(* PLC project Sin nombre, Desconocido Sin nombre 1 *)
(* stored: creationDateTime 2024-06-17T10:23:13, modificationDateTime 2024-06-20T13:18:59 *)

PROGRAM Paletizador
  VAR
    Inicio AT %IX100.0 : BOOL;
    Paro AT %IX100.1 : BOOL;
    Motor_cinta_Horizontal AT %QX100.0 : BOOL;
    Motor_cinta_Inclinado AT %QX100.1 : BOOL;
    Motor_cinta_Paletizador AT %QX100.2 : BOOL;
    Contador_Cajas AT %IX100.2 : BOOL;
    Piston_1 AT %QX100.3 : BOOL;
    Sensor_Piston_1 AT %IX100.3 : BOOL;
  END_VAR
  VAR
    CTU0 : CTU;
  END_VAR
  VAR
    Piston_Compuerta AT %QX100.4 : BOOL;
    Sensor_Piston_Compuerta AT %IX100.4 : BOOL;
    Compuerta AT %QX100.5 : BOOL;
    Sensor_Compuerta AT %IX100.5 : BOOL;
  END_VAR
  VAR
    CTU1 : CTU;
  END_VAR
  VAR
    Generador_Cajas AT %QX100.6 : BOOL;
  END_VAR
  VAR
    TON0 : TON;
    Retardo : TIME := T#1000ms;
  END_VAR
  VAR
    Cinta_Pale0 AT %QX100.7 : BOOL;
    Cinta_Pale1 AT %QX100.8 : BOOL;
    Generador_pales AT %QX100.9 : BOOL;
    Cinta_Paletizador AT %QX100.10 : BOOL;
    Sensor_Pale_0 AT %IX100.6 : BOOL;
    Sensor_Pale_1 AT %IX100.7 : BOOL;
    limite_altura AT %QX100.12 : BOOL;
    subir_pale AT %QX100.11 : BOOL;
    bajar_pale AT %QX100.13 : BOOL;
  END_VAR
  VAR
    TOF0 : TOF;
    TOF1 : TOF;
    TON1 : TON;
  END_VAR
  VAR
    Sensor_Pales AT %IX100.8 : BOOL;
    sensor_ascensor AT %IX100.9 : BOOL;
  END_VAR
  VAR
    CTU2 : CTU;
    TON2 : TON;
  END_VAR
  VAR
    sensor_bajada AT %IX100.10 : BOOL;
  END_VAR
  VAR
    TON3 : TON;
    TOF2 : TOF;
    TON4 : TON;
  END_VAR
  VAR  (* added by the conversion: wires and edge detectors of the diagram *)
    R_TRIG1 : R_TRIG;
    R_TRIG2 : R_TRIG;
    R_TRIG3 : R_TRIG;
    R_TRIG4 : R_TRIG;
    R_TRIG5 : R_TRIG;
  END_VAR

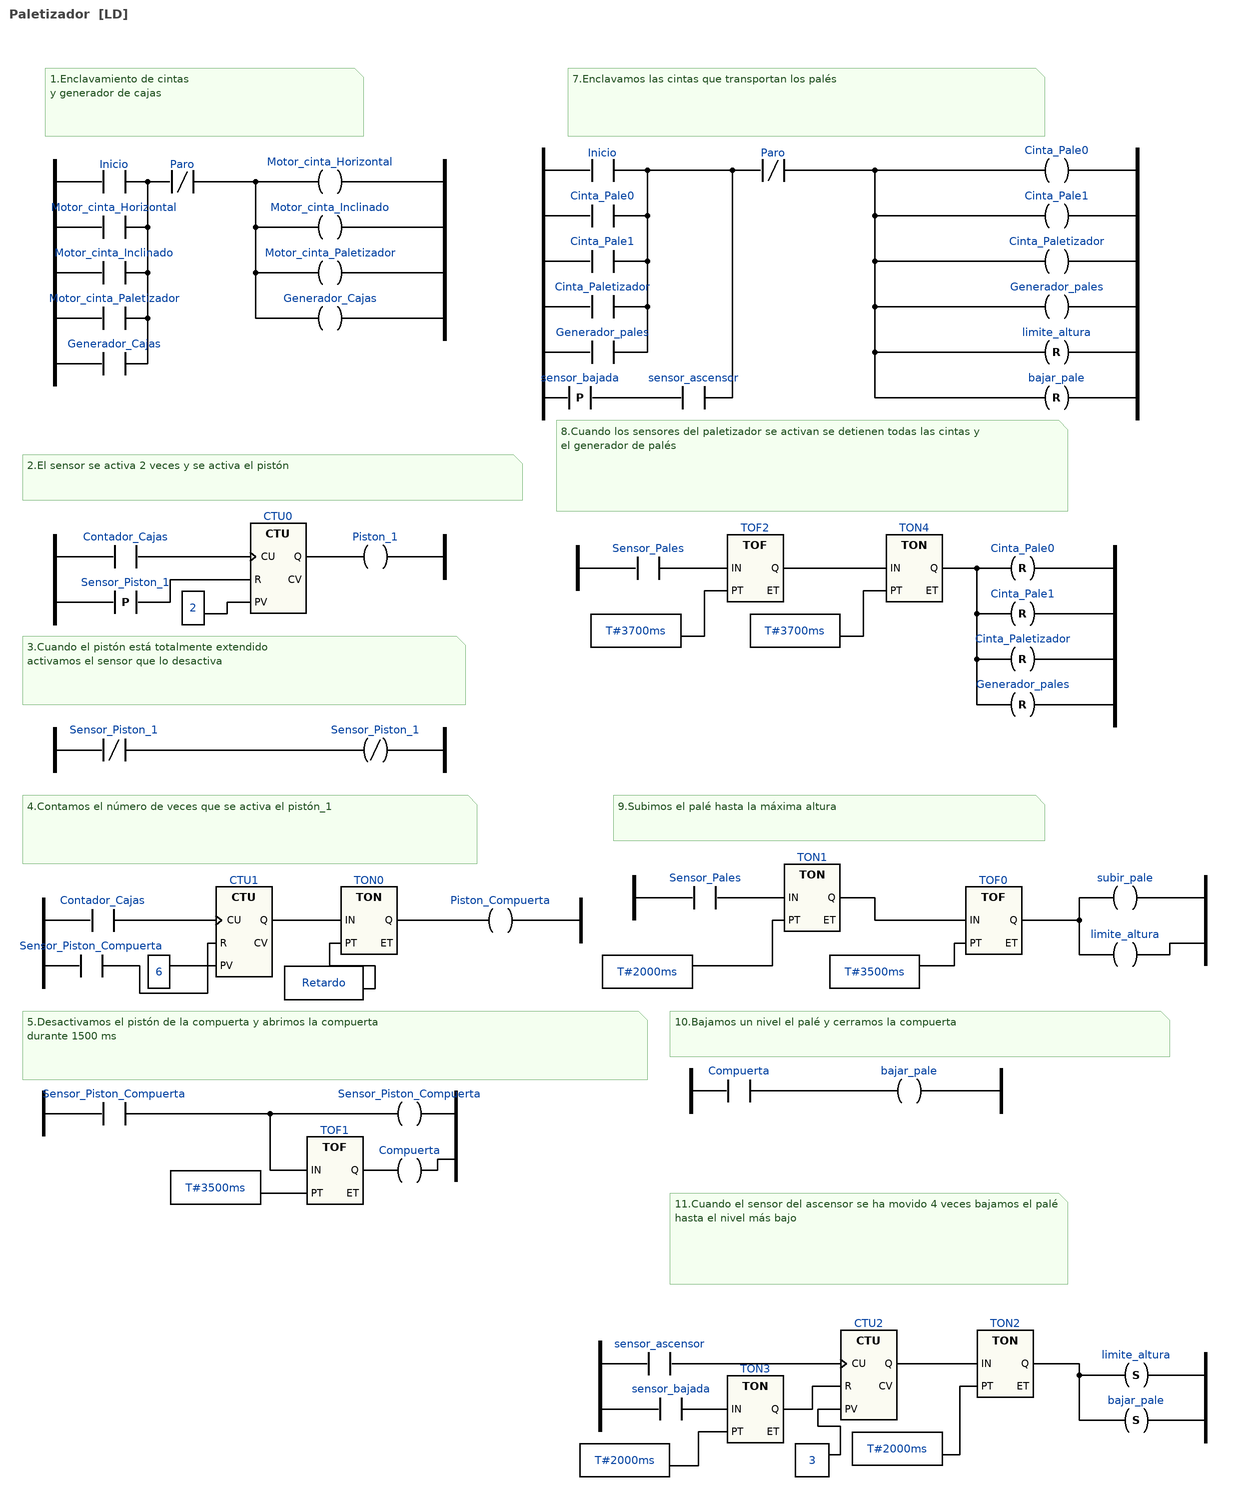
(* LD diagram, written out as Structured Text *)
(* 1.Enclavamiento de cintas
y generador de cajas *)
(* 7.Enclavamos las cintas que transportan los palés *)
Motor_cinta_Horizontal := (Inicio OR Motor_cinta_Horizontal OR Motor_cinta_Inclinado OR Motor_cinta_Paletizador OR Generador_Cajas) AND NOT Paro;
Motor_cinta_Inclinado := (Inicio OR Motor_cinta_Horizontal OR Motor_cinta_Inclinado OR Motor_cinta_Paletizador OR Generador_Cajas) AND NOT Paro;
Motor_cinta_Paletizador := (Inicio OR Motor_cinta_Horizontal OR Motor_cinta_Inclinado OR Motor_cinta_Paletizador OR Generador_Cajas) AND NOT Paro;
(* 8.Cuando los sensores del paletizador se activan se detienen todas las cintas y 
el generador de palés *)
(* 2.El sensor se activa 2 veces y se activa el pistón *)
R_TRIG1(CLK := Contador_Cajas);
R_TRIG2(CLK := Sensor_Piston_1);
CTU0(CU := R_TRIG1.Q, R := R_TRIG2.Q, PV := 2);
Piston_1 := CTU0.Q;
(* 3.Cuando el pistón está totalmente extendido
activamos el sensor que lo desactiva *)
(* 4.Contamos el número de veces que se activa el pistón_1 *)
(* 9.Subimos el palé hasta la máxima altura *)
R_TRIG3(CLK := Contador_Cajas);
CTU1(CU := R_TRIG3.Q, R := Sensor_Piston_Compuerta, PV := 6);
TON0(IN := CTU1.Q, PT := Retardo);
Piston_Compuerta := TON0.Q;
(* 5.Desactivamos el pistón de la compuerta y abrimos la compuerta
durante 1500 ms *)
(* 10.Bajamos un nivel el palé y cerramos la compuerta *)
Sensor_Piston_Compuerta := Sensor_Piston_Compuerta;
Generador_Cajas := (Inicio OR Motor_cinta_Horizontal OR Motor_cinta_Inclinado OR Motor_cinta_Paletizador OR Generador_Cajas) AND NOT Paro;
Sensor_Piston_1 := NOT (NOT Sensor_Piston_1);
TOF1(IN := Sensor_Piston_Compuerta, PT := T#3500ms);
Compuerta := TOF1.Q;
TON1(IN := Sensor_Pales, PT := T#2000ms);
TOF0(IN := TON1.Q, PT := T#3500ms);
subir_pale := TOF0.Q;
limite_altura := TOF0.Q;
bajar_pale := Compuerta;
(* 11.Cuando el sensor del ascensor se ha movido 4 veces bajamos el palé hasta el nivel más bajo *)
R_TRIG4(CLK := sensor_ascensor);
TON3(IN := sensor_bajada, PT := T#2000ms);
CTU2(CU := R_TRIG4.Q, R := TON3.Q, PV := 3);
TON2(IN := CTU2.Q, PT := T#2000ms);
IF TON2.Q THEN limite_altura := TRUE; END_IF;
IF TON2.Q THEN bajar_pale := TRUE; END_IF;
R_TRIG5(CLK := sensor_bajada);
Cinta_Pale0 := (Inicio OR Cinta_Pale0 OR Cinta_Pale1 OR Cinta_Paletizador OR Generador_pales OR R_TRIG5.Q AND sensor_ascensor) AND NOT Paro;
Cinta_Pale1 := (Inicio OR Cinta_Pale0 OR Cinta_Pale1 OR Cinta_Paletizador OR Generador_pales OR R_TRIG5.Q AND sensor_ascensor) AND NOT Paro;
Cinta_Paletizador := (Inicio OR Cinta_Pale0 OR Cinta_Pale1 OR Cinta_Paletizador OR Generador_pales OR R_TRIG5.Q AND sensor_ascensor) AND NOT Paro;
Generador_pales := (Inicio OR Cinta_Pale0 OR Cinta_Pale1 OR Cinta_Paletizador OR Generador_pales OR R_TRIG5.Q AND sensor_ascensor) AND NOT Paro;
TOF2(IN := Sensor_Pales, PT := T#3700ms);
TON4(IN := TOF2.Q, PT := T#3700ms);
IF TON4.Q THEN Cinta_Pale0 := FALSE; END_IF;
IF TON4.Q THEN Cinta_Pale1 := FALSE; END_IF;
IF TON4.Q THEN Cinta_Paletizador := FALSE; END_IF;
IF TON4.Q THEN Generador_pales := FALSE; END_IF;
IF (Inicio OR Cinta_Pale0 OR Cinta_Pale1 OR Cinta_Paletizador OR Generador_pales OR R_TRIG5.Q AND sensor_ascensor) AND NOT Paro THEN limite_altura := FALSE; END_IF;
IF (Inicio OR Cinta_Pale0 OR Cinta_Pale1 OR Cinta_Paletizador OR Generador_pales OR R_TRIG5.Q AND sensor_ascensor) AND NOT Paro THEN bajar_pale := FALSE; END_IF;
END_PROGRAM

CONFIGURATION Config0
  RESOURCE Res0 ON PLC
    TASK task0(INTERVAL := T#20ms, PRIORITY := 0);
    PROGRAM instance0 WITH task0 : Paletizador;
  END_RESOURCE
END_CONFIGURATION
